PROGRAM MAIN
VAR
	i		: DINT;
END_VAR

FOR i := 0 TO 4 DO 
	GVL.Axes[i]();
END_FOR

END_PROGRAM

(* stored: Version 1.1.0.1, ProductVersion 3.1.4024.12
   POU MAIN: Id {4cb013e4-cfb0-4f07-b880-5768dfbb58c6}, SpecialFunc None *)
